// TIA Portal V18 export
FUNCTION "mot_limited_speed" : Void   // FC12, FBD
{ S7_Optimized_Access := 'TRUE' }
VERSION : 0.1
// stored: AutoNumber true, IsIECCheckEnabled false, SetENOAutomatically false, UDAEnableTagReadback false
   VAR_INPUT
      inverter_int : Real;
      arg_a : Real;
      arg_b_bigger : Real;
      distance_crawl : Real;
      distance_fast : Real;
      distance_stop : Real;
      speed_crawl : Real;
      speed_fast : Real;
   END_VAR
   VAR_OUTPUT
      speed : Real;
   END_VAR
   VAR_TEMP
      distance1 : Real;
      distance : Real;
      can_stop : Bool;
      norm : Real;
      speed_bef_inver : Real;
   END_VAR
BEGIN

REGION Network 1
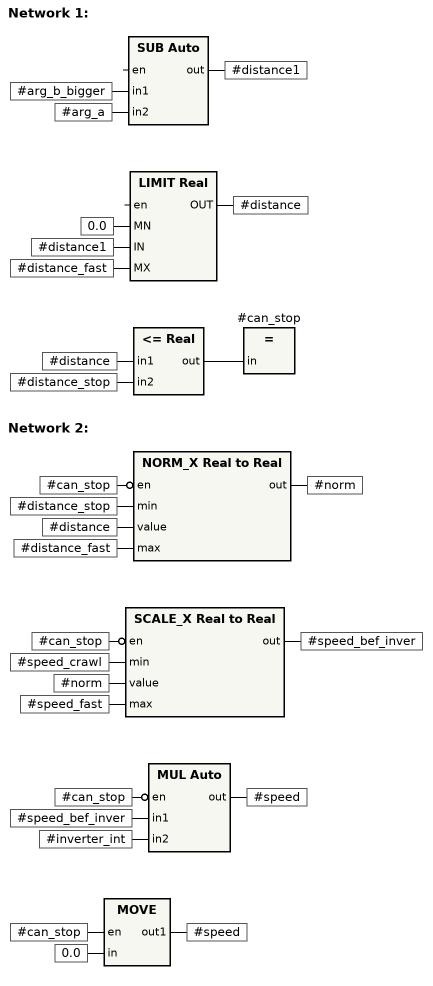
   #distance1 := #arg_b_bigger - #arg_a;
   #distance := LIMIT(MN := 0.0, IN := #distance1, MX := #distance_fast);
   #can_stop := #distance <= #distance_stop;
END_REGION

REGION Network 2
   IF NOT #can_stop THEN
       #norm := NORM_X(MIN := #distance_stop, VALUE := #distance, MAX := #distance_fast);
       #speed_bef_inver := SCALE_X(MIN := #speed_crawl, VALUE := #norm, MAX := #speed_fast);
       #speed := #speed_bef_inver * #inverter_int;
   END_IF;
   IF #can_stop THEN #speed := 0.0; END_IF;
END_REGION
END_FUNCTION
